// TIA Portal V19 export
FUNCTION_BLOCK "FeedLimiting"   // FB110, LAD
// stored: MemoryReserve 100, SetENOAutomatically true
   VAR_INPUT
      Execute { ExternalWritable := 'False'} : Bool;   // Execute Calculation
      SourceMode { ExternalWritable := 'False'} : UInt;   // Sation Work Mode
      PartLength { ExternalWritable := 'False'} : LReal;   // [mm]
      LeadCruiseVel { ExternalWritable := 'False'} : LReal;   // [mm/min]
      LeadDec { ExternalWritable := 'False'} : LReal;   // [mm/s^2]
      LeadJerk { ExternalWritable := 'False'} : LReal;   // [mm/s^3]
      ExtractionSpace { ExternalWritable := 'False'} : LReal;   // [mm]
      CarriageWorkSpace { ExternalWritable := 'False'} : LReal;   // [mm]
      Synch_Acc { ExternalWritable := 'False'} : LReal;   // [mm/s^2]
      Synch_Jerk { ExternalWritable := 'False'} : LReal;   // [mm/s^3]
      BackHomeVel { ExternalWritable := 'False'} : LReal;   // [mm/min]
      DetachVel { ExternalWritable := 'False'} : LReal;   // [mm/min]
      DetachSpace { ExternalWritable := 'False'} : LReal;   // [mm]
      CutoffTime { ExternalWritable := 'False'} : LReal;   // Cutoff Time [s]
   END_VAR
   VAR_OUTPUT
      Warning { ExternalWritable := 'False'} : Bool;
      FeedVelocity { ExternalWritable := 'False'} : LReal;   // mm/min
      ExtractionVelocity { ExternalWritable := 'False'} : LReal;
      LimitReason { ExternalWritable := 'False'} : USInt;
      Mode { ExternalWritable := 'False'} : UInt;   // Station work mode
   END_VAR
   VAR
      OldPartLength { ExternalWritable := 'False'} : LReal;
   END_VAR
   VAR RETAIN
      MaxFeedVel { ExternalVisible := 'False'; ExternalWritable := 'False'} : Struct
         PartLenth : LReal;
         CarrWS : LReal;
         Minimum : LReal;
      END_STRUCT;
   END_VAR
   VAR
      TotalGap { ExternalVisible := 'False'; ExternalWritable := 'False'} : LReal;
   END_VAR
   VAR_TEMP
      SI : Struct
         MMaxVel : LReal;
         CarriageWorkSpace : LReal;
         SAccDec : LReal;
      END_STRUCT;
      HalfPartLength : LReal;
   END_VAR
BEGIN

REGION Network 1
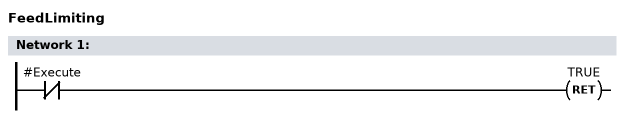
   IF NOT #Execute THEN
       ENO := TRUE;
       RETURN;
   END_IF;
END_REGION

REGION Network 2 (SCL): Unit conversion
   #SI.MMaxVel             := #LeadCruiseVel / 60000.0;

   #SI.CarriageWorkSpace   := #CarriageWorkSpace / 1000.0;

   #SI.SAccDec             := #Synch_Acc / 1000.0;
END_REGION

REGION Network 3 (SCL): Feeding max velocity due Part length
   IF  #PartLength <> #OldPartLength OR TRUE THEN
        #MaxFeedVel.PartLenth  := "VelLimitByLength"(  FeedingCruiseVel:=#LeadCruiseVel, 
                                                       PartLength:=#PartLength, 
                                                       Synch_Acc:=#Synch_Acc, 
                                                       Synch_Jerk:=#Synch_Jerk, 
                                                       BackHomeVel:=#BackHomeVel,  
                                                       Work_CycleTime:=#CutoffTime, 
                                                       DetachVel:=#DetachVel, 
                                                       DetachSpace:=#DetachSpace, 
                                                       VelTolerance:=500) / 60000.0 ;
       #OldPartLength  := #PartLength;
   END_IF;
END_REGION

REGION Network 4 (SCL): Feeding max velocity due carriage work space
   // n.b. non tiene conto dello stacco lama
   #MaxFeedVel.CarrWS :=   ( -#SI.SAccDec * #CutoffTime 
                           + SQRT_LREAL(SQR_LREAL(#SI.SAccDec)*SQR_LREAL(#CutoffTime)+4.0* #SI.SAccDec * #SI.CarriageWorkSpace)
                           ) / 2.0;
END_REGION

REGION Network 5 (SCL): Choose velocity minimum limit
   #Warning    := FALSE;
   #MaxFeedVel.Minimum := #SI.MMaxVel ;                #LimitReason   := 0;
   IF #MaxFeedVel.Minimum  > #MaxFeedVel.PartLenth THEN
       #MaxFeedVel.Minimum  := #MaxFeedVel.PartLenth;  #LimitReason   := 1;
   END_IF;
   IF #MaxFeedVel.Minimum  > #MaxFeedVel.CarrWS THEN
       #MaxFeedVel.Minimum  := #MaxFeedVel.CarrWS;     #LimitReason   := 2;
   END_IF;
END_REGION

REGION Network 6 (SCL): Choose Station work mode
   IF #SourceMode = "FS_WM_FLYING_AUTO" THEN
       // Calculate Space gap  
       #TotalGap   := "Trapezoidal_RampSpace_1"(VDelta:=#MaxFeedVel.Minimum * 60000.0, AccDec:=#LeadDec, Jerk:=#LeadJerk) + #ExtractionSpace;


       #HalfPartLength := #PartLength / 2.0;

       IF #HalfPartLength < #ExtractionSpace THEN
           #Mode           := "FS_WM_SSTILL_FWD";
           #Warning        := TRUE;
       ELSIF #HalfPartLength < #TotalGap THEN  
            #Mode           := "FS_WM_SSTILL_FWD";       
       ELSIF #HalfPartLength > #CarriageWorkSpace THEN
           #Mode           := "FS_WM_FLYING_HOME";
       ELSE 
           #Mode           := "FS_WM_FLYING_FWD";
       END_IF;

       IF #Mode = "FS_WM_SSTILL_FWD" THEN
           #MaxFeedVel.Minimum := #SI.MMaxVel ;                #LimitReason   := 0;
       END_IF;

   ELSE
       #Mode   := #SourceMode;
   END_IF;
END_REGION

REGION Network 7 (SCL): Convert output values
   #FeedVelocity       :=  #MaxFeedVel.Minimum * 60000.0;
END_REGION
END_FUNCTION_BLOCK
